TEXTLIST PML_Modes_txt
  0 = 'Undefined'
  1 = 'Production'
  2 = 'Manual'
   = ''
END_TEXTLIST

(* stored: Version 1.1.0.1, ProductVersion 3.1.4024.11
   TextList PML_Modes_txt: Id {00d82707-1059-41da-bd2b-d3b877744b83} *)
